{attribute 'GeneratedUsingTerminal: EP8309-0022-0021'}
{attribute addProperty BoxType "EP8309-0022-0021"}
{attribute addProperty Id "Reset_ErrorAT %Q*BOOL1"}
{attribute addProperty CRC "1611044825"}
{attribute addProperty Size "1"}
TYPE TACHO_Output_Channel_600697D9 :
STRUCT
	{attribute addProperty Name "Reset_Error"}
	Reset_Error AT %Q* : BOOL;
END_STRUCT
END_TYPE

(* stored: Version 1.2.0.0, ProductVersion 3.1.4024.9
   DUT TACHO_Output_Channel_600697D9: Id {91342c28-e450-4ac7-8d70-ec6e87b82966} *)
